// TIA Portal V17 export
// export: Created 2025-04-11T04:54:23.3878716Z, ExportSetting WithDefaults, DisplayName Totally Integrated Automation Portal, DisplayVersion V17, DisplayName TIA Portal Openness, DisplayVersion V17, DisplayName TIA Portal Version Control Interface, DisplayVersion V17, DisplayName SINAMICS Startdrive Advanced, DisplayVersion V17, DisplayName SINAMICS Startdrive G130, G150, S120, S150, SINAMICS MV, S210, DisplayVersion V17, DisplayName SINAMICS Startdrive G110M, G120, G120C, G120D, G120P, G115D, DisplayVersion V17, DisplayName STEP 7 Professional, DisplayVersion V17, DisplayName STEP 7 Safety, DisplayVersion V17, DisplayName WinCC Advanced, DisplayVersion V17
TYPE "用户数据类型_1"
// stored: IsFailsafeCompliant false
   STRUCT
      Element_1 { S7_SetPoint := 'True'} : Array[0..40] of "UDT_Ana_ALM";
      Element_2 { S7_SetPoint := 'True'} : Array[0..40] of "UDT_Valve_ALM";
      Element_3 { S7_SetPoint := 'True'} : Array[0..40] of "UDT_Device_ALM";
   END_STRUCT;
END_TYPE
